{attribute 'GeneratedUsingTerminal: EL3692-0000-0017'}
{attribute addProperty BoxType "EL3692-0000-0017"}
{attribute addProperty Id "SettingsAT %I*Settings_24C049402"}
{attribute addProperty CRC "3183439273"}
{attribute addProperty Size "2"}
TYPE SAI_Range_Channel_BDBF6DA9 :
STRUCT
	{attribute addProperty Name "Settings"}
	Settings AT %I* : Settings_24C04940;
END_STRUCT
END_TYPE

(* stored: Version 1.2.0.0, ProductVersion 3.1.4024.9
   DUT SAI_Range_Channel_BDBF6DA9: Id {eff1982e-0af4-4a72-a37f-01fb84b2cb03} *)
